TYPE U_Fanuc_Output :
UNION
	aStdOut		AT %Q*		:ARRAY [1..32] OF UINT;
	Control					:ST_Robot_Control;	
END_UNION
END_TYPE

(* stored: Version 1.1.0.1, ProductVersion 3.1.4024.11
   DUT U_Fanuc_Output: Id {840ff92b-13f7-4b50-9170-4952ef8224db} *)
